(* CoDeSys 2.3 export: NETVARUDPERROR.EXP *)

(* Data type *)
TYPE NetVarUDPError :
(
	NetVarUDPError_NOERROR := 0,
	NetVarUDPError_UDPSENDDATA,
	NetVarUDPError_UDPSENDACKN,
	NetVarUDPError_NOACKNOWLEDGEMENT,
	NetVarUDPError_NOTACKNOWLEDGED,
	NetVarUDPError_UDPSENDBOOTUPREQUEST,
	NetVarUDPError_UDPANSWERBOOTUPREQUEST,
	NetVarUDPError_CHECKSUM,
	NetVarUDPError_LAYOUT,

	NetVarUDPError_UDPNETWORKMANAGER_NOT_READY := 20,

	NetVarUDPError_UNKNOWN := 100
);
END_TYPE
